TYPE ST_XTS_TRANSPORT_STATE :
STRUCT
  State         : E_XTS_TRANSPORT_STATE;  // combined value of state and result(e_progress); (hint: extract state value by mod division)
  Check         : E_XTS_TRANSPORT_CHECK;

  XpuState      : ST_XPU_STATE;
  GroupInfo     : ST_GROUP_INFO; 
END_STRUCT
END_TYPE

(* stored: Version 1.1.0.1, ProductVersion 3.1.4024.12
   DUT ST_XTS_TRANSPORT_STATE: Id {926fdd85-aa28-4d62-a0b1-c60473b5d88d} *)
